PROGRAM MAIN
VAR
	fbMachine				: FB_Machine;
END_VAR

fbMachine();

END_PROGRAM

(* stored: Version 1.1.0.1, ProductVersion 3.1.4024.12
   POU MAIN: Id {97363e29-acab-41ae-b756-1e669f454fca}, SpecialFunc None *)
